Omron CX-Programmer project NewProject (CX-Programmer 9.50)

# PLC FlipFlop: CP1E E20

## Global symbols (name address type ; comment)
0.01 BOOL  ; MULAI
100.01 BOOL  ; FLIP
100.02 BOOL  ; FLOP
200.00 BOOL  ; ram
T001 BOOL  ; TDR
T002 BOOL  ; TDR2

## Program NewProgram1 (cyclic task 0)

### Section Section1

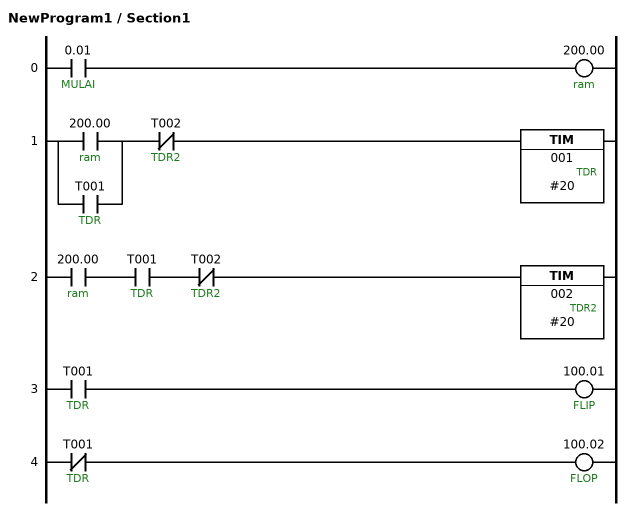
; rung 0
LD 0.01  ; MULAI
OUT 200.00  ; ram
; rung 1
LD 200.00  ; ram
OR T001  ; TDR
ANDNOT T002  ; TDR2
TIM 001 #20  ; TDR
; rung 2
LD 200.00  ; ram
AND T001  ; TDR
ANDNOT T002  ; TDR2
TIM 002 #20  ; TDR2
; rung 3
LD T001  ; TDR
OUT 100.01  ; FLIP
; rung 4
LDNOT T001  ; TDR
OUT 100.02  ; FLOP

### Section END
; rung 0
END(001)